
// ===== library: MasterCopy "Main" =====

ORGANIZATION_BLOCK "Main"   // OB1, FBD, ProgramCycle
TITLE = "Main Program Sweep (Cycle)"
{ S7_Optimized_Access := 'TRUE' }
VERSION : 0.1
   VAR_INPUT
      Initial_Call : Bool;   // Initial call of this OB
      Remanence : Bool;   // =True, if remanent data are available
   END_VAR
BEGIN

REGION Network 1
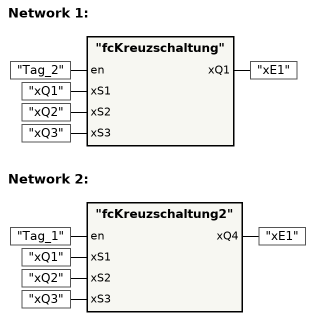
   IF "Tag_2" THEN "fcKreuzschaltung"(xS1 := "xQ1", xS2 := "xQ2", xS3 := "xQ3", xQ1 => "xE1"); END_IF;
END_REGION

REGION Network 2
   IF "Tag_1" THEN "fcKreuzschaltung2"(xS1 := "xQ1", xS2 := "xQ2", xS3 := "xQ3", xQ4 => "xE1"); END_IF;
END_REGION
END_ORGANIZATION_BLOCK

// ===== library: MasterCopy "fcKreuzschaltung" =====

FUNCTION "fcKreuzschaltung" : Void   // FC1, FBD
{ S7_Optimized_Access := 'TRUE' }
VERSION : 0.1
   VAR_INPUT
      xS1 : Bool;
      xS2 : Bool;
      xS3 : Bool;
   END_VAR
   VAR_OUTPUT
      xQ1 : Bool;
   END_VAR
BEGIN

REGION Network 1
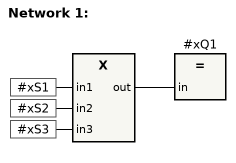
   #xQ1 := #xS1 XOR #xS2 XOR #xS3;
END_REGION
END_FUNCTION

// ===== library: MasterCopy "fcKreuzschaltung2" =====

FUNCTION "fcKreuzschaltung2" : Void   // FC2, FBD
{ S7_Optimized_Access := 'TRUE' }
VERSION : 0.1
   VAR_INPUT
      xS1 : Bool;
      xS2 : Bool;
      xS3 : Bool;
   END_VAR
   VAR_OUTPUT
      xQ4 : Bool;
   END_VAR
BEGIN

REGION Network 1
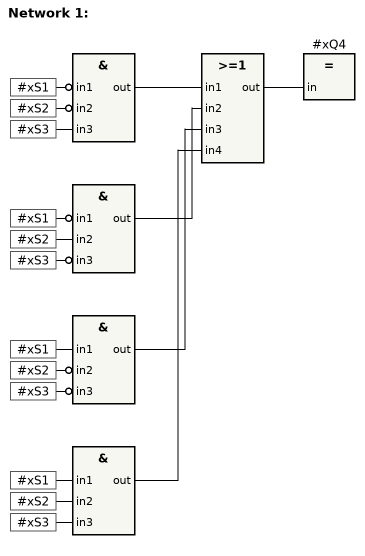
   #xQ4 := (NOT #xS1 AND NOT #xS2 AND #xS3) OR (NOT #xS1 AND #xS2 AND NOT #xS3) OR (#xS1 AND NOT #xS2 AND NOT #xS3) OR (#xS1 AND #xS2 AND #xS3);
END_REGION
END_FUNCTION

// ===== library: MasterCopy "vtKreuzschaltung" =====

VAR_GLOBAL   // PLC tag table "vtKreuzschaltung"
   "xQ1" AT %E0.0 : Bool;
   "xQ2" AT %E0.1 : Bool;
   "xQ3" AT %E0.2 : Bool;
   "xQ4" AT %A0.1 : Bool;
   "xE1" AT %A0.0 : Bool;
   "Tag_1" AT %I0.7 : Bool;
   "Tag_2" AT %I0.6 : Bool;
END_VAR

// ===== library: MasterCopy "fbstopper" =====

FUNCTION_BLOCK "fbstopper"   // FB1, FBD
{ S7_Optimized_Access := 'TRUE' }
VERSION : 0.1
   VAR_INPUT
      xAutoMode : Bool;
      xManMode : Bool;
      xQuit : Bool;
      xActStopper : Bool;
      xG1_BG9 : Bool;
      xJogDown : Bool;
      "Time 1" : Time;
      Input_1 : Bool;
   END_VAR
   VAR_OUTPUT
      xMB1 : Bool;
      xError : Bool;
   END_VAR
   VAR
      IEC_Timer_0_Instance : TON_TIME;
   END_VAR
BEGIN

REGION Network 1
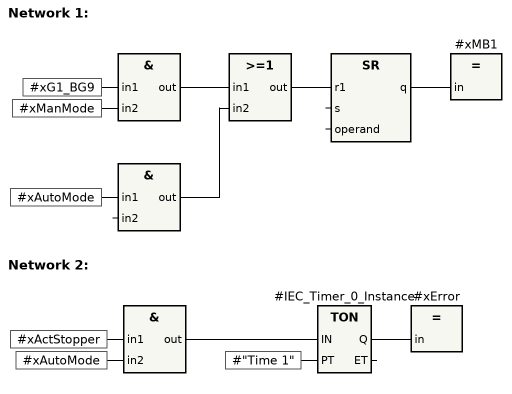
   IF (#xG1_BG9 AND #xManMode) OR #xAutoMode THEN
       <??.?> := FALSE;   // SR flip-flop
   END_IF;
   #xMB1 := <??.?>;
END_REGION

REGION Network 2
   #IEC_Timer_0_Instance(IN := #xActStopper AND #xAutoMode, PT := #"Time 1");   // TON
   #xError := #IEC_Timer_0_Instance.Q;
END_REGION
END_FUNCTION_BLOCK